# B&R Automation Studio project HealthCareDemo (part 3)

#### SemMan.cpp - SemMan Implementation
```cpp
#include "SemMan.hpp"

RouterSem::RouterSem(UDINT semaphore){
    this->_sem = semaphore;
}

//destructor
RouterSem::~RouterSem(){
    this->_type_id = rl6dNO_TYPE_ID;
}

UDINT RouterSem::get_type_id(void){
    return this->_type_id;
}
UDINT RouterSem::get_semaphore_ident(void){
    return this->_sem;
}
void RouterSem::set_delete(void){
    this->_delete = 1;
}
bool RouterSem::get_delete(void){
    return this->_delete;
}
bool RouterSem::sem_acquire(void){
    return SemAcquire(this->_sem) == ERR_OK;
}
void RouterSem::sem_release(void){
    SemRelease(this->_sem);
}
std::shared_ptr<RouterSem> RouterSem::get_shared_ptr(){
    return shared_from_this();
}

RouterSemBase::RouterSemBase(std::shared_ptr<RouterSem> router_sem){
    this->_router_semaphore = router_sem;
}

//destructor
RouterSemBase::~RouterSemBase(){
    this->_router_semaphore->set_delete();
}

bool RouterSemBase::sem_acquire(void){
    return this->_router_semaphore->sem_acquire();
}
void RouterSemBase::sem_release(void){
    this->_router_semaphore->sem_release();
}

SemMan::SemMan(){
    std::memset(&this->_create_semaphore, 0, sizeof(this->_create_semaphore));
    std::memset(&this->_delete_semaphore, 0, sizeof(this->_delete_semaphore));
}

//destructor
SemMan::~SemMan(){
    this->_type_id = rl6dNO_TYPE_ID;
}

// methods
UDINT SemMan::get_type_id(){
    return this->_type_id;
}
void SemMan::set_create_sem(){
    this->_cmd.create_sem = 1;
}
void SemMan::reset_create_sem(){
    this->_cmd.create_sem = 0;
}
std::shared_ptr<RouterSem> SemMan::get_created_sem(){
    return this->_created_semaphore;
}
bool SemMan::get_cmd_ready(){
    return this->_status.cmd_ready;
}
bool SemMan::get_done(){
    return this->_status.done;
}
bool SemMan::sem_acquire(){
    return SemAcquire(this->_sem) == ERR_OK;
}
void SemMan::sem_release(){
    SemRelease(this->_sem);
}
bool SemMan::get_initialized(){
    return this->_init_done;
}
void SemMan::cyclic(){

    switch(this->_state){

        case STATE_START:

            this->_create_semaphore.enable = 0;
            if(this->_create_semaphore.status == ERR_FUB_ENABLE_FALSE){
                this->_state = STATE_INIT;
            }

            break;

        case STATE_INIT:

            this->_create_semaphore.maxCount = 1;
            this->_create_semaphore.initCount = 1;
            this->_create_semaphore.enable = 1;
            if(this->_create_semaphore.status == ERR_OK){
                this->_sem = this->_create_semaphore.ident;
                this->_create_semaphore.enable = 0;
                this->_status.cmd_ready = 1;
                this->_init_done = 1;
                this->_state = STATE_IDLE;
            }
            else if(!((this->_create_semaphore.status == ERR_FUB_ENABLE_FALSE)||(this->_create_semaphore.status == ERR_FUB_BUSY))){
                this->_create_semaphore.enable = 0;
            }

            break;

        case STATE_IDLE:

            if(this->_cmd.delete_all){
                this->_status.cmd_ready = 0;
                // start deleting all semaphores to prepare for destruction of object
                this->_sem_iterator = this->_semaphores.begin();
                this->_state = STATE_DELETE_ALL_SEM_NEXT;
            }
            else if(this->_cmd.create_sem){
                this->_status.cmd_ready = 0;
                this->_state = STATE_CREATE_SEM;
            }
            else{
                auto it = std::find_if(this->_semaphores.begin(), this->_semaphores.end(), [](std::shared_ptr<RouterSem> i){return i->get_delete();});
                if(it != this->_semaphores.end()){
                    this->_status.cmd_ready = 0;
                    this->_sem_iterator = it;
                    std::shared_ptr<RouterSem> sem = *it;
                    this->_delete_semaphore.ident = sem->get_semaphore_ident();
                    this->_delete_semaphore.enable = 1;
                    this->_state = STATE_DELETE_SEM;
                }
            }

            break;

        case STATE_CREATE_SEM:

            this->_create_semaphore.enable = 1;

            if(this->_create_semaphore.status == ERR_OK){
                std::shared_ptr<RouterSem> new_sem (new RouterSem(this->_create_semaphore.ident));
                this->_created_semaphore = new_sem;
                this->_semaphores.push_back(new_sem);
                this->_create_semaphore.enable = 0;
                this->_status.done = 1;
                this->_state = STATE_CREATE_SEM_DONE;
            }
            else if(!((this->_create_semaphore.status == ERR_FUB_ENABLE_FALSE)||(this->_create_semaphore.status == ERR_FUB_BUSY))){
                this->_create_semaphore.enable = 0;
            }

            break;

        case STATE_CREATE_SEM_DONE:

            if(!this->_cmd.create_sem){
                this->_status.done = 0;
                this->_created_semaphore.reset();
                this->_status.cmd_ready = 1;
                this->_state = STATE_IDLE;
            }

            break;

        case STATE_DELETE_SEM:

            if(!((this->_delete_semaphore.status == ERR_FUB_ENABLE_FALSE)||(this->_delete_semaphore.status == ERR_FUB_BUSY))){
                this->_delete_semaphore.enable = 0;
                this->_semaphores.erase(this->_sem_iterator);
                this->_status.cmd_ready = 1;
                this->_state = STATE_IDLE;
            }

            break;

        case STATE_DELETE_ALL_SEM:

            if(!((this->_delete_semaphore.status == ERR_FUB_ENABLE_FALSE)||(this->_delete_semaphore.status == ERR_FUB_BUSY))){
                this->_delete_semaphore.enable = 0;
                this->_sem_iterator++;
                this->_state = STATE_DELETE_ALL_SEM_NEXT;
            }

            break;

        case STATE_DELETE_ALL_SEM_NEXT:

            if(this->_sem_iterator < this->_semaphores.end()){
                std::shared_ptr<RouterSem> sem = *this->_sem_iterator;
                this->_delete_semaphore.ident = sem->get_semaphore_ident();
                this->_delete_semaphore.enable = 1;
                this->_state = STATE_DELETE_ALL_SEM;
            }
            else{
                this->_delete_semaphore.ident = this->_sem;
                this->_delete_semaphore.enable = 1;
                this->_state = STATE_DELETE_ALL_SEM_LAST;
            }

            break;

        case STATE_DELETE_ALL_SEM_LAST:
            if(!((this->_delete_semaphore.status == ERR_FUB_ENABLE_FALSE)||(this->_delete_semaphore.status == ERR_FUB_BUSY))){
                this->_delete_semaphore.enable = 0;
                this->_semaphores.clear();
                this->_status.done = 1;
                this->_state = STATE_DELETE_ALL_SEM_DONE;
            }
            break;

        case STATE_DELETE_ALL_SEM_DONE:
            //At this point, the object must be destroyed
            break;

    }

    SemCreate(&this->_create_semaphore);
    SemDelete(&this->_delete_semaphore);

}

SemManBase::SemManBase() = default;

//destructor
SemManBase::~SemManBase() = default;

// methods
void SemManBase::set_create_sem(){
    this->_semaphore_manager.set_create_sem();
}
void SemManBase::reset_create_sem(){
    this->_semaphore_manager.reset_create_sem();
}
std::shared_ptr<RouterSem> SemManBase::get_created_sem(){
    return this->_semaphore_manager.get_created_sem();
}
bool SemManBase::get_sem_cmd_ready(){
    return this->_semaphore_manager.get_cmd_ready();
}
bool SemManBase::get_sem_done(){
    return this->_semaphore_manager.get_done();
}
bool SemManBase::sem_acquire(){
    return this->_semaphore_manager.sem_acquire();
}
void SemManBase::sem_release(){
    this->_semaphore_manager.sem_release();
}
```

#### Destination.cpp - Destination Implementation
```cpp
#include "Destination.hpp"

Destination::Destination(std::string name, std::shared_ptr<RouterSem> router_sem): RouterSemBase{router_sem}{
    this->_name = name;
}
Destination::Destination(std::string name, std::shared_ptr<RouterSem> router_sem, rl6dPositionType position): RouterSemBase{router_sem}{
    this->_name = name;
    this->_position = position;
}
Destination::Destination(std::string name, std::shared_ptr<RouterSem> router_sem, rl6dPositionType position, std::shared_ptr<Path> path_in, std::shared_ptr<Path> path_out): RouterSemBase{router_sem}{
    this->_name = name;
    this->_position = position;
    this->_path_in = path_in;
    this->_path_out = path_out;
}

//destructor
Destination::~Destination(){
    this->_type_id = rl6dNO_TYPE_ID;
}

// methods
UDINT Destination::get_type_id(){
    return this->_type_id;
}
std::string Destination::get_name(){
    return this->_name;
}
rl6dPositionType Destination::get_position(){
    return this->_position;
}
void Destination::set_position(rl6dPositionType position){
    this->_position = position;
}
std::shared_ptr<Path> Destination::get_path_in(){
    return this->_path_in;
}
void Destination::set_path_in(std::shared_ptr<Path> path){
    this->_path_in = path;
}
void Destination::clear_path_in(void){
    this->_path_in.reset();
}
std::shared_ptr<Path> Destination::get_path_out(){
    return this->_path_out;
}
void Destination::set_path_out(std::shared_ptr<Path> path){
    this->_path_out = path;
}
void Destination::clear_path_out(){
    this->_path_out.reset();
}
void Destination::set_waypoint(std::weak_ptr<Waypoint> waypoint){
    this->_waypoint = waypoint;
}
std::weak_ptr<Waypoint> Destination::get_waypoint(){
    return this->_waypoint;
}
void Destination::reset_waypoint(){
    this->_waypoint.reset();
}
std::shared_ptr<Destination> Destination::get_shared_ptr(){
    return shared_from_this();
}
std::shared_ptr<DestinationIf> Destination::create_interface(){
    std::shared_ptr<DestinationIf> destination_if (new DestinationIf);
    this->_interfaces.push_back(destination_if);
    return destination_if;
}
void Destination::add_recovery_position(rl6dPositionType position){
    this->_recovery_positions.push_back(position);
}
std::vector<rl6dPositionType> Destination::get_recovery_positions(){
    return this->_recovery_positions;
}
void Destination::set_shuttle_present(std::weak_ptr<Shuttle> shuttle){
    this->_shuttle = shuttle;
    this->_shuttle_present = 1;
}
void Destination::cyclic(){

    if(this->_shuttle_present){
        if(this->sem_acquire()){
            for(auto & interface : this->_interfaces){
                interface->set_shuttle_present(this->_shuttle);
            }
            this->sem_release();
            this->_shuttle_present = 0;
            this->_shuttle.reset();
        }
    }

    if(this->sem_acquire()){
        auto it = std::find_if(this->_interfaces.begin(), this->_interfaces.end(), [](std::shared_ptr<DestinationIf> i){return i->get_delete();});
            if(it != this->_interfaces.end()){
            this->_interfaces.erase(it);
        }
        this->sem_release();
    }

}
```

#### DestinationIf.cpp - DestinationIf Implementation
```cpp
#include "DestinationIf.hpp"

DestinationIf::DestinationIf() = default;

//destructor
DestinationIf::~DestinationIf(){
    this->_type_id = rl6dNO_TYPE_ID;
}

// methods
UDINT DestinationIf::get_type_id(){
    return this->_type_id;
}
std::shared_ptr<DestinationIf> DestinationIf::get_shared_ptr(){
    return shared_from_this();
}
void DestinationIf::set_shuttle_present(std::weak_ptr<Shuttle> shuttle){
    this->_shuttle = shuttle;
    this->_shuttle_present = 1;
}
bool DestinationIf::shuttle_is_present(void){
    return this->_shuttle_present;
}
void DestinationIf::acknowledge_shuttle(){
    this->_shuttle.reset();
    this->_shuttle_present = 0;
}
std::weak_ptr<Shuttle> DestinationIf::get_shuttle_present(){
    return this->_shuttle;
}
void DestinationIf::set_delete(){
    this->_delete = 1;
}
bool DestinationIf::get_delete(){
    return this->_delete;
}
```

#### Path.cpp - Path Implementation
```cpp
#include "Path.hpp"

Path::Path(std::string name, std::shared_ptr<RouterSem> router_sem) : RouterSemBase{router_sem}{
    this->_name = name;
}

//destructor
Path::~Path(){
    this->_type_id = rl6dNO_TYPE_ID;
}

// methods
UDINT Path::get_type_id(){
    return this->_type_id;
}
void Path::add_position(rl6dPositionType position){
    this->_positions.push_back(position);
}
std::string Path::get_name(){
    return this->_name;
}
std::shared_ptr<Path> Path::get_shared_ptr(){
    return shared_from_this();
}
std::vector<rl6dPositionType> Path::get_positions(){
    return this->_positions;
}
```

#### Waypoint.cpp - Waypoint Implementation
```cpp
#include "Waypoint.hpp"

Waypoint::Waypoint(std::string name, std::shared_ptr<RouterSem> router_sem) : RouterSemBase{router_sem}{
    this->_name = name;
}
Waypoint::Waypoint(std::string name, std::shared_ptr<RouterSem> router_sem, rl6dPositionType position) : RouterSemBase{router_sem}{
    this->_name = name;
    this->_position = position;
}

//destructor
Waypoint::~Waypoint(){
    this->_type_id = rl6dNO_TYPE_ID;
}

// methods
UDINT Waypoint::get_type_id(){
    return this->_type_id;
}
std::string Waypoint::get_name(){
    return this->_name;
}
std::shared_ptr<Waypoint> Waypoint::get_shared_ptr(){
    return shared_from_this();
}
void Waypoint::add_destination(std::shared_ptr<Destination> destination, std::shared_ptr<Path> departure_path){
    WaypointDestination waypoint_destination = {destination, departure_path};
    this->_destinations.push_back(waypoint_destination);
}
std::vector<WaypointDestination> Waypoint::get_destinations(void){
    return this->_destinations;
}
rl6dPositionType Waypoint::get_position(void){
    return this->_position;
}
std::weak_ptr<Waypoint> Waypoint::get_next_waypoint(void){
    return this->_next_waypoint;
}
void Waypoint::set_next_waypoint(std::weak_ptr<Waypoint> waypoint){
    this->_next_waypoint = waypoint;
}
void Waypoint::reset_next_waypoint(void){
    this->_next_waypoint.reset();
}
bool Waypoint::check_destination_accessible(std::shared_ptr<Destination> destination){
    for (auto & accessible_destination : this->_destinations){
        if(accessible_destination.destination == destination){
            return true;
        }
    }
    return false;
}
std::shared_ptr<Path> Waypoint::get_destination_departure_path(std::shared_ptr<Destination> destination){
    std::shared_ptr<Path> path;
    auto it = std::find_if(this->_destinations.begin(), this->_destinations.end(), [destination](WaypointDestination i){return i.destination == destination;});
    if(it != this->_destinations.end()){
        path = it->departure_path;
    }
    return path;
}
```

#### Shuttle.cpp - Shuttle Implementation
```cpp
#include "Shuttle.hpp"
ShuttleRoutePositionGenerator::ShuttleRoutePositionGenerator(){
    std::memset(&this->position, 0, sizeof(this->position));
    this->_previous_destination.reset();
    this->_next_destination.reset();
    this->_route_waypoint.reset();
    this->_current_waypoint.reset();
    this->_departure_path.reset();
}
ShuttleRoutePositionGenerator::ShuttleRoutePositionGenerator(std::shared_ptr<Destination> previous_destination, std::shared_ptr<Destination> next_destination){
    std::memset(&this->position, 0, sizeof(this->position));
    this->_previous_destination = previous_destination;
    this->_next_destination = next_destination;
    this->_route_waypoint.reset();
    this->_current_waypoint.reset();
    this->_departure_path.reset();
}
ShuttleRoutePositionGenerator::ShuttleRoutePositionGenerator(std::shared_ptr<Destination> previous_destination, std::shared_ptr<Destination> next_destination, std::weak_ptr<Waypoint> route_waypoint){
    std::memset(&this->position, 0, sizeof(this->position));
    this->_previous_destination = previous_destination;
    this->_next_destination = next_destination;
    this->_route_waypoint = route_waypoint;
    this->_current_waypoint.reset();
    this->_departure_path.reset();
}

ShuttleRoutePositionGenerator::~ShuttleRoutePositionGenerator() = default;

set_path_status_enum ShuttleRoutePositionGenerator::_set_path(std::shared_ptr<Path> path){
    this->_path = path;
    if(this->_path){
        if(this->_path->sem_acquire()){
            this->_path_positions = this->_path->get_positions();
            this->_path->sem_release();
            this->_path_iterator = this->_path_positions.begin();
            if(this->_path_iterator == this->_path_positions.end()){
                return set_path_status_invalid;
            }
            else{
                return set_path_status_valid;
            }
        }
        else{
            return set_path_status_wait_sem;
        }
    }
    else{
        return set_path_status_invalid;
    }
}

bool ShuttleRoutePositionGenerator::operator++(int){

    std::shared_ptr<Waypoint> waypoint;
    rl6dPositionType position;

    if(this->_phase == ROUTED_MOVE_PHASE_EXIT_DEST_START){
        //PHASE_EXIT_DEST_START: Attempt to get the exit path

        if(this->_previous_destination){
            this->_exit_path_status = this->_set_path(this->_previous_destination->get_path_out());
            if(this->_exit_path_status == set_path_status_valid){
                this->position.X = this->_path_iterator->X;
                this->position.Y = this->_path_iterator->Y;
                this->_path_iterator++;
                this->_phase = ROUTED_MOVE_PHASE_EXIT_DEST;
                this->event.path = this->_path;
                this->event.waypoint.reset();
                this->event.event = ROUTED_MOVE_EVENT_PATH_START;
                return true;
            }
            else if(this->_exit_path_status == set_path_status_wait_sem){
                this->event.path.reset();
                this->event.waypoint.reset();
                this->event.event = ROUTED_MOVE_EVENT_NONE;
                return false;
            }
        }
        this->_phase = ROUTED_MOVE_PHASE_WAYPOINT_START; //There is no exit path

    }
    if(this->_phase == ROUTED_MOVE_PHASE_EXIT_DEST){
        //PHASE_EXIT_DEST: Follow the exit path

        if(this->_path_iterator < this->_path_positions.end()){
            this->position.X = this->_path_iterator->X;
            this->position.Y = this->_path_iterator->Y;
            this->_path_iterator++;
            this->event.path.reset();
            this->event.waypoint.reset();
            this->event.event = ROUTED_MOVE_EVENT_NONE;
            return true;
        }
        this->_phase = ROUTED_MOVE_PHASE_WAYPOINT_START; //There are no points left on the exit path

    }
    if(this->_phase == ROUTED_MOVE_PHASE_WAYPOINT_START){
        //PHASE_WAYPOINT_START: Attempt to get the waypoint

        if(!this->_route_waypoint.expired()){
            this->_current_waypoint = this->_route_waypoint;
        }
        else if(this->_previous_destination){
            this->_current_waypoint = this->_previous_destination->get_waypoint();
        }
        if(!this->_current_waypoint.expired()){
            waypoint = this->_current_waypoint.lock();
            position = waypoint->get_position();
            this->position.X = position.X;
            this->position.Y = position.Y;
            this->_phase = ROUTED_MOVE_PHASE_WAYPOINT;
            this->event.path.reset();
            this->event.waypoint = this->_current_waypoint;
            this->event.event = ROUTED_MOVE_EVENT_WAYPOINT;
            return true;
        }
        this->_phase = ROUTED_MOVE_PHASE_ENTER_DEST_START; //There is no waypoint

    }
    if(this->_phase == ROUTED_MOVE_PHASE_WAYPOINT){
        //PHASE_WAYPOINT: Follow waypoints

        if(!this->_current_waypoint.expired()){
            waypoint = this->_current_waypoint.lock();
            if(waypoint->sem_acquire()){
                bool destination_accessible = waypoint->check_destination_accessible(this->_next_destination);
                if(destination_accessible){
                    this->_departure_path = waypoint->get_destination_departure_path(this->_next_destination);
                    waypoint->sem_release();
                    this->_phase = ROUTED_MOVE_PHASE_DEPART_WAYPOINT_START;
                }
                else{
                    waypoint->sem_release();
                    this->_current_waypoint = waypoint->get_next_waypoint();
                    if(!this->_current_waypoint.expired()){
                        waypoint = this->_current_waypoint.lock();
                        position = waypoint->get_position();
                        this->position.X = position.X;
                        this->position.Y = position.Y;
                        this->event.path.reset();
                        this->event.waypoint = this->_current_waypoint;
                        this->event.event = ROUTED_MOVE_EVENT_WAYPOINT;
                        return true;
                    }
                }
            }
            else{
                this->event.path.reset();
                this->event.waypoint.reset();
                this->event.event = ROUTED_MOVE_EVENT_NONE;
                return false;
            }
        }
        else{
            //Something went wrong here - the waypoint should not be expired
            this->_phase = ROUTED_MOVE_PHASE_ENTER_DEST_START;
        }

    }
    if(this->_phase == ROUTED_MOVE_PHASE_DEPART_WAYPOINT_START){
        //PHASE_DEPART_WAYPOINT_START: Attempt to get the departure path

        this->_departure_path_status = this->_set_path(this->_departure_path);
        if(this->_departure_path_status == set_path_status_valid){
            this->position.X = this->_path_iterator->X;
            this->position.Y = this->_path_iterator->Y;
            this->_path_iterator++;
            this->_phase = ROUTED_MOVE_PHASE_DEPART_WAYPOINT;
            this->event.path = this->_path;
            this->event.waypoint.reset();
            this->event.event = ROUTED_MOVE_EVENT_PATH_START;
            return true;
        }
        else if(this->_departure_path_status == set_path_status_wait_sem){
            this->event.path.reset();
            this->event.waypoint.reset();
            this->event.event = ROUTED_MOVE_EVENT_NONE;
            return false;
        }
        this->_phase = ROUTED_MOVE_PHASE_ENTER_DEST_START; //There is no departure path

    }
    if(this->_phase == ROUTED_MOVE_PHASE_DEPART_WAYPOINT){
        //PHASE_DEPART_WAYPOINT_START: Follow the departure path

        if(this->_departure_path_status == set_path_status_valid){
            if(this->_path_iterator < this->_path_positions.end()){
                this->position.X = this->_path_iterator->X;
                this->position.Y = this->_path_iterator->Y;
                this->_path_iterator++;
                this->event.path.reset();
                this->event.waypoint.reset();
                this->event.event = ROUTED_MOVE_EVENT_NONE;
                return true;
            }
        }
        this->_phase = ROUTED_MOVE_PHASE_ENTER_DEST_START; //There are no points left on the departure path

    }
    if(this->_phase == ROUTED_MOVE_PHASE_ENTER_DEST_START){
        //ROUTED_MOVE_PHASE_ENTER_DEST_START: Attempt to get the entry path

        this->_entry_path_status = this->_set_path(this->_next_destination->get_path_in());
        if(this->_entry_path_status == set_path_status_valid){
            this->position.X = this->_path_iterator->X;
            this->position.Y = this->_path_iterator->Y;
            this->_path_iterator++;
            this->_phase = ROUTED_MOVE_PHASE_ENTER_DEST;
            this->event.path = this->_path;
            this->event.waypoint.reset();
            this->event.event = ROUTED_MOVE_EVENT_PATH_START;
            return true;
        }
        else if(this->_entry_path_status == set_path_status_wait_sem){
            this->event.path.reset();
            this->event.waypoint.reset();
            this->event.event = ROUTED_MOVE_EVENT_NONE;
            return false;
        }
        this->_phase = ROUTED_MOVE_PHASE_DEST; //There is no entry path

    }
    if(this->_phase == ROUTED_MOVE_PHASE_ENTER_DEST){
        //ROUTED_MOVE_PHASE_ENTER_DEST: Follow the entry path

        if(this->_entry_path_status == set_path_status_valid){
            if(this->_path_iterator < this->_path_positions.end()){
                this->position.X = this->_path_iterator->X;
                this->position.Y = this->_path_iterator->Y;
                this->_path_iterator++;
                this->event.path.reset();
                this->event.waypoint.reset();
                this->event.event = ROUTED_MOVE_EVENT_NONE;
                return true;
            }
        }
        this->_phase = ROUTED_MOVE_PHASE_DEST; //There are no points left on the entry path

    }
    if(this->_phase == ROUTED_MOVE_PHASE_DEST){
        //ROUTED_MOVE_PHASE_DEST: Move to destination

        position = this->_next_destination->get_position();
        this->position.X = position.X;
        this->position.Y = position.Y;
        if(this->_updated_destination){
            this->_previous_destination = this->_next_destination;
            this->_next_destination = this->_updated_destination;
            this->_updated_destination.reset();
            this->_phase = ROUTED_MOVE_PHASE_EXIT_DEST_START;
        }
        else{
            this->_done = 1;
            this->_phase = ROUTED_MOVE_PHASE_ARRIVE;
        }
        this->event.path.reset();
        this->event.waypoint.reset();
        this->event.event = ROUTED_MOVE_EVENT_NONE;
        return true;

    }

    return false;

}

void ShuttleRoutePositionGenerator::update_destination(std::shared_ptr<Destination> destination){
    if(this->_phase < ROUTED_MOVE_PHASE_DEPART_WAYPOINT_START){ //We have not yet left for the current destination
        this->_next_destination = destination;
    }
    else{
        this->_updated_destination = destination;
    }
}

void ShuttleRoutePositionGenerator::update_destination(std::shared_ptr<Destination> destination, std::weak_ptr<Waypoint> waypoint){
    if(!waypoint.expired()){
        this->_route_waypoint = waypoint;
    }
    if(this->_phase < ROUTED_MOVE_PHASE_DEPART_WAYPOINT_START){ //We have not yet left for the current destination
        this->_next_destination = destination;
    }
    else{
        this->_updated_destination = destination;
    }
}

routed_move_phase_enum ShuttleRoutePositionGenerator::get_phase(){
    return this->_phase;
}
bool ShuttleRoutePositionGenerator::get_done(){
    return this->_done;
}

Shuttle::Shuttle(Mc6DShuttleType shuttle, std::shared_ptr<RouterSem> router_sem, UDINT user_data_size, UINT shuttle_id) : RouterSemBase{router_sem}{
    std::memset(&this->_move_in_plane, 0, sizeof(this->_move_in_plane));
    this->_shuttle = shuttle;
    this->_move_in_plane.Shuttle = &this->_shuttle;
    this->_move_in_plane.Parameters.Mode = mcACP6D_MOVE_ABSOLUTE;
    this->_user_data = std::unique_ptr<char[]>(new char[user_data_size]);
    std::memset(this->_user_data.get(), 0, user_data_size);
    this->_user_data_size = user_data_size;
    this->_shuttle_id = shuttle_id;
}

//destructor
Shuttle::~Shuttle(){
    this->_type_id = rl6dNO_TYPE_ID;
}

// methods
UDINT Shuttle::get_type_id(){
    return this->_type_id;
}
UINT Shuttle::get_shuttle_id(){
    return this->_shuttle_id;
}
Mc6DShuttleType* Shuttle::get_shuttle_reference(){
    return &this->_shuttle;
}
std::shared_ptr<Destination> Shuttle::get_current_destination(){
    return this->_next_destination;
}
std::shared_ptr<Destination> Shuttle::get_previous_destination(){
    return this->_previous_destination;
}
void Shuttle::clear_previous_destination(){
    this->_previous_destination.reset();
}
std::shared_ptr<ShuttleIf> Shuttle::create_interface(){
    std::shared_ptr<ShuttleIf> shuttle_if (new ShuttleIf);
    this->_interfaces.push_back(shuttle_if);
    return shuttle_if;
}
std::shared_ptr<Shuttle> Shuttle::get_shared_ptr(){
    return shared_from_this();
}
ReadUserDataResult Shuttle::read_user_data(){
    ReadUserDataResult result = {this->_user_data.get(), this->_user_data_size};
    return result;
}
UDINT Shuttle::write_user_data(char* value, UDINT size){
    if(size < this->_user_data_size){
        std::memcpy(this->_user_data.get(), value, size);
        return size;
    }
    else{
        std::memcpy(this->_user_data.get(), value, this->_user_data_size);
        return this->_user_data_size;
    }
}
bool Shuttle::_update_interfaces(){
    if(this->_current_interface){
        if(this->_interfaces.empty()){ //The current interface is defined, but no interfaces are being used
            this->_current_interface.reset();
            return 1; //Indicate that the interface has changed
        }
        else if(this->_current_interface != this->_interfaces.back()){ //A newer interface is available
            std::shared_ptr<ShuttleIf> interface = this->_current_interface;
            interface->reset_move_active();
            interface->set_aborted();
            this->_current_interface = this->_interfaces.back();
            return 1; //Indicate that the interface has changed
        }
    }
    else if(!this->_interfaces.empty()){ //No interface is defined, but an interface is available
        this->_current_interface = this->_interfaces.back();
        return 1; //Indicate that the interface has changed
    }
    return 0; //Indicate that the interface has not changed
}

void Shuttle::_log_event(RoutedMoveEvent event){

    switch(event.event){

        case ROUTED_MOVE_EVENT_NONE:

            break;

        case ROUTED_MOVE_EVENT_PATH_START:
            log_path_start(this->get_shuttle_id(), this->_route_position_generator.event.path->get_name());
            break;

        case ROUTED_MOVE_EVENT_WAYPOINT:
            log_waypoint_move(this->get_shuttle_id(), this->_route_position_generator.event.waypoint.lock()->get_name());
            break;

    }

    return;

}

void Shuttle::cyclic(){

    rl6dPositionType position;

    switch(this->_state){

        case STATE_IDLE:

            if(this->_update_interfaces()){
                if(this->_current_interface){
                    this->_move_in_plane.Parameters.Velocity = this->_current_interface->get_velocity();
                    this->_move_in_plane.Parameters.Acceleration = this->_current_interface->get_acceleration();
                    this->_current_interface->set_move_active();
                    this->_next_destination = this->_current_interface->get_destination();
                    if(this->_current_interface->get_destination_direct_command()){
                        position = this->_next_destination->get_position();
                        this->_move_in_plane.Parameters.Position.X = position.X;
                        this->_move_in_plane.Parameters.Position.Y = position.Y;
                        this->_move_in_plane.Execute = 1;
                        log_direct_move_start(this->get_shuttle_id(), this->_next_destination->get_name());
                        this->_state = STATE_DIRECT_MOVE;
                    }
                    else if(this->_current_interface->get_destination_command()){
                        this->_optional_waypoint = this->_current_interface->get_waypoint();
                        this->_route_position_generator = ShuttleRoutePositionGenerator(this->_previous_destination, this->_next_destination, this->_optional_waypoint);
                        if(this->_route_position_generator++){
                            this->_move_in_plane.Parameters.Position.X = _route_position_generator.position.X;
                            this->_move_in_plane.Parameters.Position.Y = _route_position_generator.position.Y;
                            this->_move_in_plane.Execute = 1;
                            if(this->_optional_waypoint.expired()){
                                log_routed_move_start(this->get_shuttle_id(), this->_next_destination->get_name());
                            }
                            else{
                                log_routed_move_waypoint(this->get_shuttle_id(), this->_next_destination->get_name(), this->_optional_waypoint.lock()->get_name());
                            }
                            this->_log_event(this->_route_position_generator.event);
                            this->_state = STATE_ROUTED_MOVE;
                        }
                        else{
                            this->_state = STATE_ROUTED_MOVE_START;
                        }
                    }
                }
            }

            break;

        case STATE_ROUTED_MOVE_START:

            if(this->_route_position_generator++){
                this->_move_in_plane.Parameters.Position.X = _route_position_generator.position.X;
                this->_move_in_plane.Parameters.Position.Y = _route_position_generator.position.Y;
                this->_move_in_plane.Execute = 1;
                if(this->_optional_waypoint.expired()){
                    log_routed_move_start(this->get_shuttle_id(), this->_next_destination->get_name());
                }
                else{
                    log_routed_move_waypoint(this->get_shuttle_id(), this->_next_destination->get_name(), this->_optional_waypoint.lock()->get_name());
                }
                this->_log_event(this->_route_position_generator.event);
                this->_state = STATE_ROUTED_MOVE;
            }

            break;

        case STATE_ROUTED_MOVE:

            if(this->_move_in_plane.Done){
                this->_move_in_plane.Execute = 0;
                if(this->_route_position_generator.get_done()){
                    log_destination_arrival(this->get_shuttle_id(), this->_next_destination->get_name());
                    if(this->_current_interface){
                        this->_current_interface->set_move_done();
                    }
                    std::weak_ptr<Shuttle> reference = shared_from_this();
                    this->_next_destination->set_shuttle_present(reference);
                    this->_previous_destination = this->_next_destination;
                    this->_next_destination.reset();
                    this->_state = STATE_IDLE;
                }
                else{
                    this->_state = STATE_ROUTED_MOVE_NEXT;
                }
            }
            else if(this->_move_in_plane.Error){
                log_sh_error(this->get_shuttle_id(), this->_move_in_plane.ErrorID);
                this->_move_in_plane.Execute = 0;
                this->_current_interface->set_error(this->_move_in_plane.ErrorID);
                this->_state = STATE_IDLE;
            }

            break;

        case STATE_ROUTED_MOVE_NEXT:

            if(this->_update_interfaces()){
                if(this->_current_interface){
                    this->_move_in_plane.Parameters.Velocity = this->_current_interface->get_velocity();
                    this->_move_in_plane.Parameters.Acceleration = this->_current_interface->get_acceleration();
                    this->_current_interface->set_move_active();
                    this->_next_destination = this->_current_interface->get_destination();
                    this->_route_position_generator.update_destination(this->_next_destination);
                    log_destination_update(this->get_shuttle_id(), this->_next_destination->get_name());
                }
            }
            if(this->_route_position_generator++){
                this->_move_in_plane.Parameters.Position.X = _route_position_generator.position.X;
                this->_move_in_plane.Parameters.Position.Y = _route_position_generator.position.Y;
                this->_move_in_plane.Execute = 1;
                this->_log_event(this->_route_position_generator.event);
                this->_state = STATE_ROUTED_MOVE;
            }

            break;

        case STATE_DIRECT_MOVE:

            if(this->_move_in_plane.Done){
                this->_move_in_plane.Execute = 0;
                log_destination_arrival(this->get_shuttle_id(), this->_next_destination->get_name());
                if(this->_current_interface){
                    this->_current_interface->set_move_done();
                }
                std::weak_ptr<Shuttle> reference = shared_from_this();
                this->_next_destination->set_shuttle_present(reference);
                this->_previous_destination = this->_next_destination;
                this->_next_destination.reset();
                this->_state = STATE_IDLE;
            }
            else if(this->_move_in_plane.Error){
                log_sh_error(this->get_shuttle_id(), this->_move_in_plane.ErrorID);
                this->_move_in_plane.Execute = 0;
                if(this->_current_interface){
                    this->_current_interface->set_error(this->_move_in_plane.ErrorID);
                }
                this->_state = STATE_IDLE;
            }

            break;

    }

    if(this->sem_acquire()){
        auto it_delete = std::find_if(this->_interfaces.begin(), this->_interfaces.end(), [](std::shared_ptr<ShuttleIf> i){return i->get_delete();});
        if(it_delete != this->_interfaces.end()){
            this->_interfaces.erase(it_delete);
        }
        //Delete any invalid interfaces
        auto it_invalid = std::find_if(this->_interfaces.begin(), this->_interfaces.end(), [](std::shared_ptr<ShuttleIf> i){return (i->get_type_id() != rl6dSHUTTLE_IF_TYPE_ID);});
        if(it_invalid != this->_interfaces.end()){
            this->_interfaces.erase(it_invalid);
        }
        this->sem_release();
    }

    MC_BR_MoveInPlane_Acp6D(&this->_move_in_plane);

}
```

#### ShuttleIf.cpp - DestinationIf Implementation
```cpp
#include "ShuttleIf.hpp"

ShuttleIf::ShuttleIf() = default;

//destructor
ShuttleIf::~ShuttleIf(){
    this->_type_id = rl6dNO_TYPE_ID;
}

// methods
UDINT ShuttleIf::get_type_id(){
    return this->_type_id;
}
void ShuttleIf::set_destination(std::shared_ptr<Destination> destination, REAL velocity, REAL acceleration){
    this->_destination = destination;
    this->_velocity = velocity;
    this->_acceleration = acceleration;
    this->_move_destination = 1;
}
bool ShuttleIf::get_destination_command(){
    return this->_move_destination;
}
void ShuttleIf::set_destination_direct(std::shared_ptr<Destination> destination, REAL velocity, REAL acceleration){
    this->_destination = destination;
    this->_velocity = velocity;
    this->_acceleration = acceleration;
    this->_move_destination_direct = 1;
}
bool ShuttleIf::get_destination_direct_command(){
    return this->_move_destination_direct;
}
std::shared_ptr<Destination> ShuttleIf::get_destination(){
    return this->_destination;
}
void ShuttleIf::set_aborted(){
    this->_aborted = 1;
}
bool ShuttleIf::get_aborted(){
    return this->_aborted;
}
void ShuttleIf::set_error(DINT error){
    this->_error = 1;
    this->_error_id = error;
}
bool ShuttleIf::get_error(){
    return this->_error;
}
DINT ShuttleIf::get_error_id(){
    return this->_error_id;
}
void ShuttleIf::set_move_done(){
    this->_move_done = 1;
}
bool ShuttleIf::get_move_done(){
    return this->_move_done;
}
void ShuttleIf::set_move_active(){
    this->_move_active = 1;
}
void ShuttleIf::reset_move_active(){
    this->_move_active = 0;
}
bool ShuttleIf::get_move_active(){
    return this->_move_active;
}
void ShuttleIf::set_delete(){
    this->_delete = 1;
}
bool ShuttleIf::get_delete(){
    return this->_delete;
}
REAL ShuttleIf::get_velocity(){
    return this->_velocity;
}
REAL ShuttleIf::get_acceleration(){
    return this->_acceleration;
}
std::shared_ptr<ShuttleIf> ShuttleIf::get_shared_ptr(){
    return shared_from_this();
}
```

#### rl6dRouterMan.cpp - rl6dRouter Implementation
```cpp
#include "Router.hpp"

uint32_t bur_heap_size = rl6dHEAP_SIZE;

extern "C" _BUR_PUBLIC void rl6dRouterMan(struct rl6dRouterMan* inst){

    if(inst == nullptr){
        return;
    }

    Router* r;
    DINT error;

    enum state{
        state_idle,
        state_active,
        state_error
    };

    switch(inst->Internal.State){

        case state_idle:

            if(inst->Enable){
                inst->Busy = 1;
                if(inst->UserDataSize > 0){
                    inst->Router.Ident = reinterpret_cast<std::uintptr_t>(new Router(inst->Assembly, inst->UserDataSize));
                    inst->Active = 1;
                    inst->Internal.State = state_active;
                }
                else{
                    inst->ErrorID = rl6dERR_USER_DATA_SIZE_ZERO;
                    inst->Error = 1;
                    inst->Internal.State = state_error;
                }
            }

            break;

        case state_active:

            error = check_router_reference(&inst->Router);
            if(error == ERR_OK){
                r = reinterpret_cast<Router*>(inst->Router.Ident);
                r->cyclic();
                if(!inst->Enable){
                    inst->Active = 0;
                    inst->Router.Ident = 0;
                    delete r;
                    inst->Busy = 0;
                    inst->Internal.State = state_idle;
                    }
            }
            else{
                inst->Active = 0;
                inst->ErrorID = error;
                inst->Error = 1;
                inst->Internal.State = state_error;
            }

            break;

        case state_error:

            if(!inst->Enable){
                error = check_router_reference(&inst->Router);
                if(error == ERR_OK){
                    r = reinterpret_cast<Router*>(inst->Router.Ident);
                    delete r;
                }
                inst->Router.Ident = 0;
                inst->ErrorID = ERR_OK;
                inst->Error = 0;
                inst->Busy = 0;
                inst->Internal.State = state_idle;
            }

            break;

    }

    //TODO: Allow for cleanup of semaphores before router deletion

}
```

#### rl6dRouterAddPathFromData.cpp - rl6dRouterAddPathFromData Implementation
```cpp
#include "Router.hpp"

extern "C" _BUR_PUBLIC void rl6dRouterAddPathFromData(struct rl6dRouterAddPathFromData* inst){

    if(inst == nullptr){
        return;
    }

    Router* r;
    RouterSem* router_sem;
    std::shared_ptr<Path> p;
    rl6dPositionType* position;
    DINT error;

    enum state{
        state_idle,
        state_create_sem_start,
        state_create_sem_end,
        state_add_positions,
        state_done,
        state_error
    };

    switch(inst->Internal.State){

        case state_idle:

            if(inst->Execute){
                inst->Busy = 1;
                inst->Internal.State = state_create_sem_start;
            }

            break;

        case state_create_sem_start:

            error = check_router_reference(inst->Router);
            if(error == ERR_OK){
                if(inst->DataSize % sizeof(rl6dPositionType) != 0){
                    error = rl6dERR_DATA_ALIGNMENT;
                }
            }
            if(error == ERR_OK){
                if(inst->Name[0] == 0){
                    error = rl6dERR_NO_OBJ_NAME;
                }
            }
            if(error == ERR_OK){
                r = reinterpret_cast<Router*>(inst->Router->Ident);
                if(r->get_initialized()){
                    if(r->sem_acquire()){
                        if(r->get_sem_cmd_ready()){
                            r->set_create_sem();
                            inst->Internal.State = state_create_sem_end;
                        }
                        else{
                            r->sem_release();
                        }
                    }
                }
            }
            else{
                inst->ErrorID = error;
                inst->Error = 1;
                inst->Internal.State = state_error;
            }
            break;

        case state_create_sem_end:

            error = check_router_reference(inst->Router);
            if(error == ERR_OK){
                r = reinterpret_cast<Router*>(inst->Router->Ident);
                if(r->get_sem_done()){
                    inst->Internal.Reference = reinterpret_cast<std::uintptr_t>(r->get_created_sem().get());
                    r->reset_create_sem();
                    r->sem_release();
                    inst->Internal.State = state_add_positions;
                }
            }
            else{
                inst->ErrorID = error;
                inst->Error = 1;
                inst->Internal.State = state_error;
            }

            break;

        case state_add_positions:

            error = check_router_reference(inst->Router);
            if(error == ERR_OK){
                error = check_router_sem_reference(inst->Internal.Reference);
            }
            if(error == ERR_OK){
                if(inst->DataSize % sizeof(rl6dPositionType) != 0){
                    error = rl6dERR_DATA_ALIGNMENT;
                }
            }
            if(error == ERR_OK){
                if(inst->Name[0] == 0){
                    error = rl6dERR_NO_OBJ_NAME;
                }
            }
            if(error == ERR_OK){
                r = reinterpret_cast<Router*>(inst->Router->Ident);
                if(r->acquire_path_semaphore()){
                    router_sem = reinterpret_cast<RouterSem*>(inst->Internal.Reference);
                    try{
                        p = r->create_path(inst->Name, router_sem->get_shared_ptr());
                    }
                    catch (const std::invalid_argument& ia) {
                        inst->ErrorID = rl6dERR_OBJ_NAME_EXISTS;
                        inst->Error = 1;
                        inst->Internal.State = state_error;
                        r->release_path_semaphore();
                        router_sem->set_delete();
                        return;
                    }
                    for(UDINT offset = 0; offset < inst->DataSize; offset += sizeof(rl6dPositionType)){
                        position = reinterpret_cast<rl6dPositionType*>(inst->DataAddress + offset);
                        p->add_position(*position);
                    }
                    inst->Path.Ident = reinterpret_cast<std::uintptr_t>(p.get());
                    r->release_path_semaphore();
                    inst->Done = 1;
                    inst->Internal.State = state_done;
                }
            }
            else{
                inst->ErrorID = error;
                inst->Error = 1;
                if(check_router_sem_reference(inst->Internal.Reference) == ERR_OK){
                    router_sem = reinterpret_cast<RouterSem*>(inst->Internal.Reference);
                    router_sem->set_delete();
                }
                inst->Internal.State = state_error;
            }

            break;

        case state_done:

            if(!inst->Execute){
                inst->Done = 0;
                inst->Path.Ident = 0;
                inst->Busy = 0;
                inst->Internal.State = state_idle;
            }

            break;

        case state_error:

            if(!inst->Execute){
                inst->ErrorID = ERR_OK;
                inst->Error = 0;
                inst->Busy = 0;
                inst->Internal.State = state_idle;
            }

            break;

    }

}
```

#### rl6dRouterAddDestination.cpp - rl6dRouterAddDestination Implementation
```cpp
#include "Router.hpp"

extern "C" _BUR_PUBLIC void rl6dRouterAddDestination(struct rl6dRouterAddDestination* inst){

    if(inst == nullptr){
        return;
    }

    Router* r;
    RouterSem* router_sem;
    std::shared_ptr<Destination> destination;
    Path* p;
    std::shared_ptr<Path> entry_path;
    std::shared_ptr<Path> exit_path;
    DINT error;

    enum state{
        state_idle,
        state_create_sem_start,
        state_create_sem_end,
        state_create_destination,
        state_done,
        state_error
    };

    switch(inst->Internal.State){

        case state_idle:

            if(inst->Execute){
                inst->Busy = 1;
                inst->Internal.State = state_create_sem_start;
            }

            break;

        case state_create_sem_start:

            error = check_router_reference(inst->Router);
            if(error == ERR_OK){
                if(inst->Name[0] == 0){
                    error = rl6dERR_NO_OBJ_NAME;
                }
            }
            if((error == ERR_OK) && (inst->EntryPath != nullptr)){
                error = check_path_reference(inst->EntryPath);
            }
            if((error == ERR_OK) && (inst->ExitPath != nullptr)){
                error = check_path_reference(inst->ExitPath);
            }
            if(error == ERR_OK){
                r = reinterpret_cast<Router*>(inst->Router->Ident);
                if(r->get_initialized()){
                    if(r->sem_acquire()){
                        if(r->get_sem_cmd_ready()){
                            r->set_create_sem();
                            inst->Internal.State = state_create_sem_end;
                        }
                        else{
                            r->sem_release();
                        }
                    }
                }
            }
            else{
                inst->ErrorID = error;
                inst->Error = 1;
                inst->Internal.State = state_error;
            }
            break;

        case state_create_sem_end:

            error = check_router_reference(inst->Router);
            if(error == ERR_OK){
                r = reinterpret_cast<Router*>(inst->Router->Ident);
                if(r->get_sem_done()){
                    inst->Internal.Reference = reinterpret_cast<std::uintptr_t>(r->get_created_sem().get());
                    r->reset_create_sem();
                    r->sem_release();
                    inst->Internal.State = state_create_destination;
                }
            }
            else{
                inst->ErrorID = error;
                inst->Error = 1;
                inst->Internal.State = state_error;
            }

            break;

        case state_create_destination:

            error = check_router_reference(inst->Router);
            if(error == ERR_OK){
            error = check_router_sem_reference(inst->Internal.Reference);
            }
            if(error == ERR_OK){
                if(inst->Name[0] == 0){
                    error = rl6dERR_NO_OBJ_NAME;
                }
            }
            if((error == ERR_OK) && (inst->EntryPath != nullptr)){
                error = check_path_reference(inst->EntryPath);
            }
            if((error == ERR_OK) && (inst->ExitPath != nullptr)){
                error = check_path_reference(inst->ExitPath);
            }
            if(error == ERR_OK){
                r = reinterpret_cast<Router*>(inst->Router->Ident);
                if(r->acquire_destination_semaphore()){
                    router_sem = reinterpret_cast<RouterSem*>(inst->Internal.Reference);
                    if(inst->EntryPath != nullptr){
                        if(inst->EntryPath->Ident){
                            p = reinterpret_cast<Path*>(inst->EntryPath->Ident);
                            if(p->get_type_id() == rl6dPATH_TYPE_ID){
                                entry_path = p->get_shared_ptr();
                            }
                        }
                    }
                    if(inst->ExitPath != nullptr){
                        if(inst->ExitPath->Ident){
                            p = reinterpret_cast<Path*>(inst->ExitPath->Ident);
                            if(p->get_type_id() == rl6dPATH_TYPE_ID){
                                exit_path = p->get_shared_ptr();
                            }
                        }
                    }
                    try{
                        destination = r->create_destination(inst->Name, router_sem->get_shared_ptr(), inst->Position, entry_path, exit_path);
                    }
                    catch (const std::invalid_argument& ia) {
                        inst->ErrorID = rl6dERR_OBJ_NAME_EXISTS;
                        inst->Error = 1;
                        inst->Internal.State = state_error;
                        r->release_destination_semaphore();
                        router_sem->set_delete();
                        return;
                    }
                    inst->Destination.Ident = reinterpret_cast<std::uintptr_t>(destination.get());
                    r->release_destination_semaphore();
                    inst->Done = 1;
                    inst->Internal.State = state_done;
                }
            }
            else{
                inst->ErrorID = error;
                inst->Error = 1;
                if(check_router_sem_reference(inst->Internal.Reference) == ERR_OK){
                    router_sem = reinterpret_cast<RouterSem*>(inst->Internal.Reference);
                    router_sem->set_delete();
                }
                inst->Internal.State = state_error;
            }

            break;

        case state_done:

            if(!inst->Execute){
                inst->Done = 0;
                inst->Destination.Ident = 0;
                inst->Busy = 0;
                inst->Internal.State = 0;
            }

            break;

        case state_error:

            if(!inst->Execute){
                inst->ErrorID = ERR_OK;
                inst->Error = 0;
                inst->Busy = 0;
                inst->Internal.State = state_idle;
            }

            break;

    }

}
```

#### rl6dRouterAddWaypoint.cpp - rl6dRouterAddWaypoint Implementation
```cpp
#include "Router.hpp"

extern "C" _BUR_PUBLIC void rl6dRouterAddWaypoint(struct rl6dRouterAddWaypoint* inst){

    if(inst == nullptr){
        return;
    }

    Router* r;
    RouterSem* router_sem;
    std::shared_ptr<Waypoint> waypoint;
    DINT error;

    enum state{
        state_idle,
        state_create_sem_start,
        state_create_sem_end,
        state_create_waypoint,
        state_done,
        state_error
    };

    switch(inst->Internal.State){

        case state_idle:

            if(inst->Execute){
                inst->Busy = 1;
                inst->Internal.State = state_create_sem_start;
            }

            break;

        case state_create_sem_start:

            error = check_router_reference(inst->Router);
            if(error == ERR_OK){
                if(inst->Name[0] == 0){
                    error = rl6dERR_NO_OBJ_NAME;
                }
            }
            if(error == ERR_OK){
                r = reinterpret_cast<Router*>(inst->Router->Ident);
                if(r->get_initialized()){
                    if(r->sem_acquire()){
                        if(r->get_sem_cmd_ready()){
                            r->set_create_sem();
                            inst->Internal.State = state_create_sem_end;
                        }
                        else{
                            r->sem_release();
                        }
                    }
                }
            }
            else{
                inst->ErrorID = error;
                inst->Error = 1;
                inst->Internal.State = state_error;
            }
            break;

        case state_create_sem_end:

            error = check_router_reference(inst->Router);
            if(error == ERR_OK){
                r = reinterpret_cast<Router*>(inst->Router->Ident);
                if(r->get_sem_done()){
                    inst->Internal.Reference = reinterpret_cast<std::uintptr_t>(r->get_created_sem().get());
                    r->reset_create_sem();
                    r->sem_release();
                    inst->Internal.State = state_create_waypoint;
                }
            }
            else{
                inst->ErrorID = error;
                inst->Error = 1;
                inst->Internal.State = state_error;
            }

            break;

        case state_create_waypoint:

            error = check_router_reference(inst->Router);
            if(error == ERR_OK){
            error = check_router_sem_reference(inst->Internal.Reference);
            }
            if(error == ERR_OK){
                if(inst->Name[0] == 0){
                    error = rl6dERR_NO_OBJ_NAME;
                }
            }
            if(error == ERR_OK){
                r = reinterpret_cast<Router*>(inst->Router->Ident);
                if(r->acquire_waypoint_semaphore()){
                    router_sem = reinterpret_cast<RouterSem*>(inst->Internal.Reference);
                    try{
                        waypoint = r->create_waypoint(inst->Name, router_sem->get_shared_ptr(), inst->Position);
                    }
                    catch (const std::invalid_argument& ia) {
                        inst->ErrorID = rl6dERR_OBJ_NAME_EXISTS;
                        inst->Error = 1;
                        inst->Internal.State = state_error;
                        r->release_waypoint_semaphore();
                        router_sem->set_delete();
                        return;
                    }
                    inst->Waypoint.Ident = reinterpret_cast<std::uintptr_t>(waypoint.get());
                    r->release_waypoint_semaphore();
                    inst->Done = 1;
                    inst->Internal.State = state_done;
                }
            }
            else{
                inst->ErrorID = error;
                inst->Error = 1;
                if(check_router_sem_reference(inst->Internal.Reference) == ERR_OK){
                    router_sem = reinterpret_cast<RouterSem*>(inst->Internal.Reference);
                    router_sem->set_delete();
                }
                inst->Internal.State = state_error;
            }

            break;

        case state_done:

            if(!inst->Execute){
                inst->Done = 0;
                inst->Waypoint.Ident = 0;
                inst->Busy = 0;
                inst->Internal.State = 0;
            }

            break;

        case state_error:

            if(!inst->Execute){
                inst->ErrorID = ERR_OK;
                inst->Error = 0;
                inst->Busy = 0;
                inst->Internal.State = state_idle;
            }

            break;

    }

}
```

#### rl6dPathGetData.cpp - rl6dGetDataFromPath Implementation
```cpp
#include "Router.hpp"

extern "C" _BUR_PUBLIC void rl6dPathGetData(struct rl6dPathGetData* inst){

    if(inst == nullptr){
        return;
    }

    Path* p;
    std::shared_ptr<Path> path;
    DINT error;

    enum state{
        state_idle,
        state_get_data,
        state_done,
        state_error
    };

    switch(inst->Internal.State){

        case state_idle:

            if(inst->Execute){
                inst->Busy = 1;
                inst->Internal.DataAddress = inst->DataAddress;
                inst->Internal.DataSize = inst->DataSize;
                inst->Internal.State = state_get_data;
            }

            break;

        case state_get_data:

            error = check_path_reference(inst->Path);
            if(error == ERR_OK){
                p = reinterpret_cast<Path*>(inst->Path->Ident);
                path = p->get_shared_ptr();
                if(path->sem_acquire()){
                    std::vector<rl6dPositionType> positions = path->get_positions();
                    path->sem_release();
                    UDINT available_size = inst->Internal.DataSize / sizeof(rl6dPositionType);
                    UDINT offset = 0;
                    for(auto & position : positions){
                        if(offset < available_size){
                            rl6dPositionType* array_position = reinterpret_cast<rl6dPositionType*>(inst->Internal.DataAddress + offset*sizeof(rl6dPositionType));
                            *array_position = position;
                            offset++;
                        }
                        else{
                            break;
                        }
                    }
                    inst->PathDataSize = positions.size() * sizeof(rl6dPositionType);
                    inst->Done = 1;
                    inst->Internal.State = state_done;
                }
            }
            else{
                inst->ErrorID = error;
                inst->Error = 1;
                inst->Internal.State = state_error;
            }

            break;

        case state_done:

            if(!inst->Execute){
                inst->Done = 0;
                std::memset(reinterpret_cast<void*>(inst->Internal.DataAddress), 0, inst->Internal.DataSize);
                inst->Busy = 0;
                inst->Internal.State = state_idle;
            }

            break;

        case state_error:

            if(!inst->Execute){
                inst->ErrorID = ERR_OK;
                inst->Error = 0;
                inst->Busy = 0;
                inst->Internal.State = state_idle;
            }

            break;

    }

}
```

#### rl6dDestAddRecoveryPosFromData.cpp - rl6dRouterAddPathFromData Implementation
```cpp
#include "Router.hpp"

extern "C" _BUR_PUBLIC void rl6dDestAddRecoveryPosFromData(struct rl6dDestAddRecoveryPosFromData* inst){

    if(inst == nullptr){
        return;
    }

    Destination* d;
    std::shared_ptr<Destination> destination;
    rl6dPositionType* position;
    DINT error;

    enum state{
        state_idle,
        state_add_recovery_pos,
        state_done,
        state_error
    };

    switch(inst->Internal.State){

        case state_idle:

            if(inst->Execute){
                inst->Busy = 1;
                inst->Internal.State = state_add_recovery_pos;
            }

            break;

        case state_add_recovery_pos:

            error = check_destination_reference(inst->Destination);
            if(error == ERR_OK){
                if(inst->DataSize % sizeof(rl6dPositionType) != 0){
                    error = rl6dERR_DATA_ALIGNMENT;
                }
            }
            if(error == ERR_OK){
                d = reinterpret_cast<Destination*>(inst->Destination->Ident);
                destination = d->get_shared_ptr();
                if(destination->sem_acquire()){
                    for(UDINT offset = 0; offset < inst->DataSize; offset += sizeof(rl6dPositionType)){
                        position = reinterpret_cast<rl6dPositionType*>(inst->DataAddress + offset);
                        destination->add_recovery_position(*position);
                    }
                    destination->sem_release();
                    inst->Done = 1;
                    inst->Internal.State = state_done;
                }
            }
            else{
                inst->ErrorID = error;
                inst->Error = 1;
                inst->Internal.State = state_error;
            }
            break;

        case state_done:

            if(!inst->Execute){
                inst->Done = 0;
                inst->Busy = 0;
                inst->Internal.State = state_idle;
            }

            break;

        case state_error:

            if(!inst->Execute){
                inst->ErrorID = ERR_OK;
                inst->Error = 0;
                inst->Busy = 0;
                inst->Internal.State = state_idle;
            }

            break;
    }

}
```

#### rl6dDestinationSetWaypoint.cpp - rl6dWaypointSetNextWaypoint Implementation
```cpp
#include "Router.hpp"

extern "C" _BUR_PUBLIC void rl6dDestinationSetWaypoint(struct rl6dDestinationSetWaypoint* inst){

    if(inst == nullptr){
        return;
    }

    Destination* d;
    std::shared_ptr<Destination> destination;
    Waypoint* w;
    DINT error;

    enum state{
        state_idle,
        state_done,
        state_error
    };

    switch(inst->Internal.State){

        case state_idle:

            if(inst->Execute){
                inst->Busy = 1;
                error = check_destination_reference(inst->Destination);
                if(error == ERR_OK){
                    error = check_waypoint_reference(inst->Waypoint);
                }
                if(error == ERR_OK){
                    d = reinterpret_cast<Destination*>(inst->Destination->Ident);
                    destination = d->get_shared_ptr();
                    w = reinterpret_cast<Waypoint*>(inst->Waypoint->Ident);
                    destination->set_waypoint(w->get_shared_ptr());
                    inst->Done = 1;
                    inst->Internal.State = state_done;
                }
                else{
                    inst->ErrorID = error;
                    inst->Error = 1;
                    inst->Internal.State = state_error;
                }
            }

            break;

        case state_done:

            if(!inst->Execute){
                inst->Done = 0;
                inst->Busy = 0;
                inst->Internal.State = state_idle;
            }

            break;

        case state_error:

            if(!inst->Execute){
                inst->ErrorID = ERR_OK;
                inst->Error = 0;
                inst->Busy = 0;
                inst->Internal.State = state_idle;
            }

            break;
    }

}
```

#### rl6dWaypointAddDestination.cpp - rl6dWaypointAddDestination Implementation
```cpp
#include "Router.hpp"

extern "C" _BUR_PUBLIC void rl6dWaypointAddDestination(struct rl6dWaypointAddDestination* inst){

    if(inst == nullptr){
        return;
    }

    Waypoint* w;
    std::shared_ptr<Waypoint> waypoint;
    Destination* d;
    Path* p;
    std::shared_ptr<Path> path;
    DINT error;

    enum state{
        state_idle,
        state_add_destination,
        state_done,
        state_error
    };

    switch(inst->Internal.State){

        case state_idle:

            if(inst->Execute){
                inst->Busy = 1;
                inst->Internal.State = state_add_destination;
            }

            break;

        case state_add_destination:

            error = check_waypoint_reference(inst->Waypoint);
            if(error == ERR_OK){
                error = check_destination_reference(inst->Destination);
            }
            if((error == ERR_OK) && (inst->DeparturePath != nullptr)){
                error = check_path_reference(inst->DeparturePath);
            }
            if(error == ERR_OK){
                w = reinterpret_cast<Waypoint*>(inst->Waypoint->Ident);
                waypoint = w->get_shared_ptr();
                if(waypoint->sem_acquire()){
                    if(inst->DeparturePath != nullptr){
                        p = reinterpret_cast<Path*>(inst->Waypoint->Ident);
                        path = p->get_shared_ptr();
                    }
                    d = reinterpret_cast<Destination*>(inst->Destination->Ident);
                    waypoint->add_destination(d->get_shared_ptr(), path);
                    waypoint->sem_release();
                    inst->Done = 1;
                    inst->Internal.State = state_done;
                }
            }
            else{
                inst->ErrorID = error;
                inst->Error = 1;
                inst->Internal.State = state_error;
            }
            break;

        case state_done:

            if(!inst->Execute){
                inst->Done = 0;
                inst->Busy = 0;
                inst->Internal.State = state_idle;
            }

            break;

        case state_error:

            if(!inst->Execute){
                inst->ErrorID = ERR_OK;
                inst->Error = 0;
                inst->Busy = 0;
                inst->Internal.State = state_idle;
            }

            break;
    }

}
```

#### rl6dWaypointSetNextWaypoint.cpp - rl6dWaypointSetNextWaypoint Implementation
```cpp
#include "Router.hpp"

extern "C" _BUR_PUBLIC void rl6dWaypointSetNextWaypoint(struct rl6dWaypointSetNextWaypoint* inst){

    if(inst == nullptr){
        return;
    }

    Waypoint* w;
    std::shared_ptr<Waypoint> waypoint;
    Waypoint* w_n;
    DINT error;

    enum state{
        state_idle,
        state_done,
        state_error
    };

    switch(inst->Internal.State){

        case state_idle:

            if(inst->Execute){
                inst->Busy = 1;
                error = check_waypoint_reference(inst->Waypoint);
                if(error == ERR_OK){
                    error = check_waypoint_reference(inst->NextWaypoint);
                }
                if(error == ERR_OK){
                    w = reinterpret_cast<Waypoint*>(inst->Waypoint->Ident);
                    waypoint = w->get_shared_ptr();
                    w_n = reinterpret_cast<Waypoint*>(inst->NextWaypoint->Ident);
                    waypoint->set_next_waypoint(w_n->get_shared_ptr());
                    inst->Done = 1;
                    inst->Internal.State = state_done;
                }
                else{
                    inst->ErrorID = error;
                    inst->Error = 1;
                    inst->Internal.State = state_error;
                }
            }

            break;

        case state_done:

            if(!inst->Execute){
                inst->Done = 0;
                inst->Busy = 0;
                inst->Internal.State = state_idle;
            }

            break;

        case state_error:

            if(!inst->Execute){
                inst->ErrorID = ERR_OK;
                inst->Error = 0;
                inst->Busy = 0;
                inst->Internal.State = state_idle;
            }

            break;
    }

}
```

#### rl6dRouterAddShFromAsm.cpp - rl6dRouterAddShFromAsm Implementation
```cpp
#include "Router.hpp"

extern "C" _BUR_PUBLIC void rl6dRouterAddShFromAsm(struct rl6dRouterAddShFromAsm* inst){

    if(inst == nullptr){
        return;
    }

    Router* r;
    DINT error;

    enum state{
        state_idle,
        state_send_cmd,
        state_add_shuttles,
        state_done,
        state_error
    };

    switch(inst->Internal.State){

        case state_idle:

            if(inst->Execute){
                inst->Busy = 1;
                inst->Internal.State = state_send_cmd;
            }

            break;

        case state_send_cmd:

            error = check_router_reference(inst->Router);
            if(error == ERR_OK){
                r = reinterpret_cast<Router*>(inst->Router->Ident);
                if(r->get_initialized()){
                    if(r->acquire_cmd_semaphore()){
                        if(r->get_cmd_ready()){
                            r->set_add_sh_from_asm();
                            inst->Internal.State = state_add_shuttles;
                        }
                        else{
                            r->release_cmd_semaphore();
                        }
                    }
                }
            }
            else{
                inst->ErrorID  = error;
                inst->Error = 1;
                inst->Internal.State = state_error;
            }

            break;

        case state_add_shuttles:

            error = check_router_reference(inst->Router);
            if(error == ERR_OK){
                r = reinterpret_cast<Router*>(inst->Router->Ident);
                if(r->get_done()){
                    inst->NumShuttles = r->get_num_asm_sh();
                    r->reset_add_sh_from_asm();
                    r->release_cmd_semaphore();
                    inst->Done = 1;
                    inst->Internal.State = state_done;
                }
                else if(r->get_error()){
                    r->reset_add_sh_from_asm();
                    inst->ErrorID  = r->get_error_id();
                    inst->Error = 1;
                    r->set_error_reset();
                    r->release_cmd_semaphore();
                    inst->Internal.State = state_error;
                }
            }
            else{
                inst->ErrorID  = error;
                inst->Error = 1;
                inst->Internal.State = state_error;
            }

            break;

        case state_done:

            if(!inst->Execute){
                inst->Done = 0;
                inst->Busy = 0;
                inst->NumShuttles = 0;
                inst->Internal.State = state_idle;
            }

            break;

        case state_error:

            if(!inst->Execute){
                inst->ErrorID = ERR_OK;
                inst->Error = 0;
                inst->Busy = 0;
                inst->Internal.State = state_idle;
            }

            break;

    }

}
```

#### rl6dRouterExecuteRecovery.cpp - rl6dRouterExecuteRecovery Implementation
```cpp
#include "Router.hpp"

extern "C" _BUR_PUBLIC void rl6dRouterExecuteRecovery(struct rl6dRouterExecuteRecovery* inst){

    if(inst == nullptr){
        return;
    }

    Router* r;
    DINT error;

    enum state{
        state_idle,
        state_send_cmd,
        state_recover,
        state_done,
        state_error
    };

    switch(inst->Internal.State){

        case state_idle:

            if(inst->Execute){
                inst->Busy = 1;
                inst->Internal.State = state_send_cmd;
            }

            break;

        case state_send_cmd:

            error = check_router_reference(inst->Router);
            if(error == ERR_OK){
                r = reinterpret_cast<Router*>(inst->Router->Ident);
                if(r->get_initialized()){
                    if(r->acquire_cmd_semaphore()){
                        if(r->get_cmd_ready()){
                            r->set_recover_shuttles(inst->Mode, inst->Velocity, inst->Acceleration);
                            inst->Internal.State = state_recover;
                        }
                        else{
                            r->release_cmd_semaphore();
                        }
                    }
                }
            }
            else{
                inst->ErrorID  = error;
                inst->Error = 1;
                inst->Internal.State = state_error;
            }

            break;

        case state_recover:

            error = check_router_reference(inst->Router);
            if(error == ERR_OK){
                r = reinterpret_cast<Router*>(inst->Router->Ident);
                if(r->get_done()){
                    r->reset_recover_shuttles();
                    r->release_cmd_semaphore();
                    inst->Done = 1;
                    inst->Internal.State = state_done;
                }
                else if(r->get_error()){
                    r->reset_recover_shuttles();
                    inst->ErrorID  = r->get_error_id();
                    inst->Error = 1;
                    r->set_error_reset();
                    r->release_cmd_semaphore();
                    inst->Internal.State = state_error;
                }
            }
            else{
                inst->ErrorID  = error;
                inst->Error = 1;
                inst->Internal.State = state_error;
            }

            break;

        case state_done:

            if(!inst->Execute){
                inst->Done = 0;
                inst->Busy = 0;
                inst->Internal.State = state_idle;
            }

            break;

        case state_error:

            if(!inst->Execute){
                inst->ErrorID = ERR_OK;
                inst->Error = 0;
                inst->Busy = 0;
                inst->Internal.State = state_idle;
            }

            break;

    }

}
```

#### rl6dDestinationMonitor.cpp - rl6dDestinationMonitor Implementation
```cpp
#include "Router.hpp"

extern "C" _BUR_PUBLIC void rl6dDestinationMonitor(struct rl6dDestinationMonitor* inst){

    if(inst == nullptr){
        return;
    }

    Destination* d;
    std::shared_ptr<Destination> destination;
    DestinationIf* i;
    std::shared_ptr<DestinationIf> interface;
    std::shared_ptr<Shuttle> shuttle;
    DINT error;

    enum state{
        state_idle,
        state_get_interface,
        state_wait_shuttle,
        state_wait_not_acknowledge,
        state_wait_acknowledge,
        state_error
    };

    switch(inst->Internal.State){

        case state_idle:

            if(inst->Enable){
                inst->Busy = 1;
                inst->Internal.State = state_get_interface;
            }

            break;

        case state_get_interface:

            error = check_destination_reference(inst->Destination);
            if(error == ERR_OK){
                d = reinterpret_cast<Destination*>(inst->Destination->Ident);
                destination = d->get_shared_ptr();
                if(destination->sem_acquire()){
                    inst->Internal.Reference = reinterpret_cast<std::uintptr_t>(destination->create_interface().get());
                    destination->sem_release();
                    inst->Internal.State = state_wait_shuttle;
                }
            }
            else{
                inst->ErrorID = error;
                inst->Error = 1;
                inst->Internal.State = state_error;
            }

            break;

        case state_wait_shuttle:

            error = check_destination_if_reference(inst->Internal.Reference);
            if(error == ERR_OK){
                if(inst->Enable){
                    i = reinterpret_cast<DestinationIf*>(inst->Internal.Reference);
                    interface = i->get_shared_ptr();
                    if(interface->shuttle_is_present()){
                        shuttle = interface->get_shuttle_present().lock();
                        inst->ShuttleID = shuttle->get_shuttle_id();
                        inst->RouterShuttle.Ident = reinterpret_cast<std::uintptr_t>(shuttle.get());
                        inst->Mc6DShuttle = *shuttle->get_shuttle_reference();
                        inst->ShuttlePresent = 1;
                        interface->acknowledge_shuttle();
                        if(inst->AcknowledgeShuttle){
                            inst->Internal.State = state_wait_not_acknowledge;
                        }
                        else{
                            inst->Internal.State = state_wait_acknowledge;
                        }
                    }
                    inst->Valid = 1;
                }
                else{
                    i = reinterpret_cast<DestinationIf*>(inst->Internal.Reference);
                    interface = i->get_shared_ptr();
                    interface->set_delete();
                    inst->Valid = 0;
                    inst->ShuttlePresent = 0;
                    inst->ShuttleID = 0;
                    std::memset(&inst->Mc6DShuttle, 0, sizeof(inst->Mc6DShuttle));
                    std::memset(&inst->RouterShuttle, 0, sizeof(inst->RouterShuttle));
                    inst->Busy = 0;
                    inst->Internal.State = state_idle;
                }
            }
            else{
                inst->ErrorID = error;
                inst->Error = 1;
                inst->Internal.State = state_error;
            }

            break;

        case state_wait_not_acknowledge:

            if(inst->Enable){
                if(!inst->AcknowledgeShuttle){
                    inst->Internal.State = state_wait_acknowledge;
                }
            }
            else{
                error = check_destination_if_reference(inst->Internal.Reference);
                if(error == ERR_OK){
                    i = reinterpret_cast<DestinationIf*>(inst->Internal.Reference);
                    interface = i->get_shared_ptr();
                    interface->set_delete();
                    inst->Valid = 0;
                    inst->ShuttlePresent = 0;
                    inst->ShuttleID = 0;
                    std::memset(&inst->Mc6DShuttle, 0, sizeof(inst->Mc6DShuttle));
                    std::memset(&inst->RouterShuttle, 0, sizeof(inst->RouterShuttle));
                    inst->Busy = 0;
                    inst->Internal.State = state_idle;
                }
                else{
                    inst->Valid = 0;
                    inst->ShuttlePresent = 0;
                    inst->ShuttleID = 0;
                    std::memset(&inst->Mc6DShuttle, 0, sizeof(inst->Mc6DShuttle));
                    std::memset(&inst->RouterShuttle, 0, sizeof(inst->RouterShuttle));
                    inst->ErrorID = error;
                    inst->Error = 1;
                    inst->Internal.State = state_error;
                }
            }

            break;

        case state_wait_acknowledge:

            if(inst->Enable){
                if(inst->AcknowledgeShuttle){
                    inst->ShuttlePresent = 0;
                    inst->ShuttleID = 0;
                    std::memset(&inst->Mc6DShuttle, 0, sizeof(inst->Mc6DShuttle));
                    std::memset(&inst->RouterShuttle, 0, sizeof(inst->RouterShuttle));
                    inst->Internal.State = state_wait_shuttle;
                }
            }
            else{
                error = check_destination_if_reference(inst->Internal.Reference);
                if(error == ERR_OK){
                    i = reinterpret_cast<DestinationIf*>(inst->Internal.Reference);
                    interface = i->get_shared_ptr();
                    interface->set_delete();
                    inst->Valid = 0;
                    inst->ShuttlePresent = 0;
                    inst->ShuttleID = 0;
                    std::memset(&inst->Mc6DShuttle, 0, sizeof(inst->Mc6DShuttle));
                    std::memset(&inst->RouterShuttle, 0, sizeof(inst->RouterShuttle));
                    inst->Busy = 0;
                    inst->Internal.State = state_idle;
                }
                else{
                    inst->Valid = 0;
                    inst->ShuttlePresent = 0;
                    inst->ShuttleID = 0;
                    std::memset(&inst->Mc6DShuttle, 0, sizeof(inst->Mc6DShuttle));
                    std::memset(&inst->RouterShuttle, 0, sizeof(inst->RouterShuttle));
                    inst->ErrorID = error;
                    inst->Error = 1;
                    inst->Internal.State = state_error;
                }
            }

            break;

        case state_error:

            if(!inst->Enable){
                inst->ErrorID = ERR_OK;
                inst->Error = 0;
                inst->Busy = 0;
                inst->Internal.State = state_idle;
            }

            break;

    }

}
```

#### rl6dShuttleMoveDestination.cpp - rl6dDestinationMonitor Implementation
```cpp
#include "Router.hpp"

extern "C" _BUR_PUBLIC void rl6dShuttleMoveDestination(struct rl6dShuttleMoveDestination* inst){

    if(inst == nullptr){
        return;
    }

    Destination* d;
    std::shared_ptr<Destination> destination;
    Waypoint* w;
    std::weak_ptr<Waypoint> waypoint;
    Shuttle* s;
    std::shared_ptr<Shuttle> shuttle;
    ShuttleIf* i;
    std::shared_ptr<ShuttleIf> interface;
    DINT error;

    enum state{
        state_idle,
        state_send_cmd,
        state_move,
        state_done,
        state_error
    };

    switch(inst->Internal.State){

        case state_idle:

            if(inst->Execute){
                inst->Busy = 1;
                inst->Internal.State = state_send_cmd;
            }

            break;

        case state_send_cmd:

            error = check_shuttle_reference(inst->RouterShuttle);
            if(error == ERR_OK){
                error = check_destination_reference(inst->Destination);
            }
            if(error == ERR_OK){
                s = reinterpret_cast<Shuttle*>(inst->RouterShuttle->Ident);
                shuttle = s->get_shared_ptr();
                if(shuttle->sem_acquire()){
                    inst->Internal.Reference = reinterpret_cast<std::uintptr_t>(shuttle->create_interface().get());
                    shuttle->sem_release();
                    d = reinterpret_cast<Destination*>(inst->Destination->Ident);
                    destination = d->get_shared_ptr();
                    error = check_shuttle_if_reference(inst->Internal.Reference);
                    if(error == ERR_OK){
                        i = reinterpret_cast<ShuttleIf*>(inst->Internal.Reference);
                        interface = i->get_shared_ptr();
                        if (inst->Waypoint != nullptr){
                            error = check_waypoint_reference(inst->Waypoint);
                            if(error == ERR_OK){
                                w = reinterpret_cast<Waypoint*>(inst->Waypoint->Ident);
                                waypoint = w->get_shared_ptr();
                                interface->set_destination_waypoint(destination, waypoint, inst->Velocity, inst->Acceleration);
                                inst->Internal.State = state_move;
                            }
                            else{
                                inst->ErrorID = error;
                                inst->Error = 1;
                                inst->Internal.State = state_error;
                            }
                        }
                        else{
                            interface->set_destination(destination, inst->Velocity, inst->Acceleration);
                            inst->Internal.State = state_move;
                        }
                    }
                    else{
                        inst->ErrorID = error;
                        inst->Error = 1;
                        inst->Internal.State = state_error;
                    }
                }
            }
            else{
                inst->ErrorID = error;
                inst->Error = 1;
                inst->Internal.State = state_error;
            }

            break;

        case state_move:

            error = check_shuttle_if_reference(inst->Internal.Reference);
            if(error == ERR_OK){
                i = reinterpret_cast<ShuttleIf*>(inst->Internal.Reference);
                interface = i->get_shared_ptr();
                if(inst->Execute){
                    if(interface->get_error()){
                        inst->ErrorID = interface->get_error_id();
                        inst->Error = 1;
                        inst->Active = 0;
                        inst->Aborted = 0;
                        inst->Done = 0;
                        inst->Internal.State = state_error;
                    }
                    else{
                        inst->Active = interface->get_move_active();
                        inst->Aborted = interface->get_aborted();
                        inst->Done = interface->get_move_done();
                    }
                }
                else{
                    inst->Active = 0;
                    inst->Aborted = 0;
                    inst->Done = 0;
                    interface->set_delete();
                    inst->Internal.Reference = 0;
                    inst->Busy = 0;
                    inst->Internal.State = state_idle;
                }
            }
            else{
                inst->Active = 0;
                inst->Aborted = 0;
                inst->Done = 0;
                inst->ErrorID = error;
                inst->Error = 1;
                inst->Internal.State = state_error;
            }

            break;

        case state_error:

            if(!inst->Execute){
                error = check_shuttle_if_reference(inst->Internal.Reference);
                if(error == ERR_OK){
                    interface->set_delete();
                    inst->Internal.Reference = 0;
                }
                inst->ErrorID = ERR_OK;
                inst->Error = 0;
                inst->Busy = 0;
                inst->Internal.State = state_idle;
            }

            break;

    }

}
```

#### rl6dShCopyUserData.cpp - rl6dShCopyUserData Implementation
```cpp
#include "Shuttle.hpp"
#include "CheckRef.hpp"

extern "C" _BUR_PUBLIC void rl6dShCopyUserData(struct rl6dShCopyUserData* inst){

    if(inst == nullptr){
        return;
    }

    Shuttle* s;
    std::shared_ptr<Shuttle> shuttle;
    DINT error;

    enum state{
        state_idle,
        state_done,
        state_error
    };

    switch(inst->Internal.State){

        case state_idle:

            if(inst->Execute){
                inst->Busy = 1;
                error = check_shuttle_reference(inst->RouterShuttle);
                if(error == ERR_OK){
                    if(inst->DataAddress == 0){
                        error = rl6dERR_USER_DATA_NULL_POINTER;
                    }
                }
                if(error == ERR_OK){
                    if(inst->DataSize == 0){
                        error = rl6dERR_USER_DATA_SIZE_ZERO;
                    }
                }
                if(error == ERR_OK){
                    s = reinterpret_cast<Shuttle*>(inst->RouterShuttle->Ident);
                    shuttle = s->get_shared_ptr();
                    ReadUserDataResult result = shuttle->read_user_data();
                    if(result.size == inst->DataSize){
                        if(inst->Mode == rl6dSH_COPY_USER_DATA_READ){
                            std::memcpy(reinterpret_cast<char*>(inst->DataAddress), result.value, result.size);
                            inst->SizeCopied = result.size;
                        }
                        else if(inst->Mode == rl6dSH_COPY_USER_DATA_WRITE){
                            inst->SizeCopied = shuttle->write_user_data(reinterpret_cast<char*>(inst->DataAddress), inst->DataSize);
                        }
                        inst->Done = 1;
                        inst->Internal.State = state_done;
                    }
                    else{
                        inst->ErrorID = rl6dERR_USER_DATA_SIZE_MISMATCH;
                        inst->Error = 1;
                        inst->Internal.State = state_error;
                    }
                }
                else{
                    inst->ErrorID = error;
                    inst->Error = 1;
                    inst->Internal.State = state_error;
                }
            }

            break;

        case state_done:

            if(!inst->Execute){
                inst->Done = 0;
                inst->SizeCopied = 0;
                inst->Busy = 0;
                inst->Internal.State = state_idle;
            }

            break;

        case state_error:

            if(!inst->Execute){
                inst->ErrorID = ERR_OK;
                inst->Error = 0;
                inst->Busy = 0;
                inst->Internal.State = state_idle;
            }

            break;

    }

}
```

#### rl6dShCopyUserDataSync.cpp - rl6dShCopyUserDataSync Implementation
```cpp
#include "Shuttle.hpp"
#include "CheckRef.hpp"

extern "C" _BUR_PUBLIC signed long rl6dShCopyUserDataSync(struct rl6dShuttleType* RouterShuttle, enum rl6dShCopyUserDataModeEnum Mode, unsigned long DataAddress, unsigned long DataSize){

    Shuttle* s;
    std::shared_ptr<Shuttle> shuttle;
    DINT error;

    error = check_shuttle_reference(RouterShuttle);
    if(error == ERR_OK){
        if(DataAddress == 0){
            error = rl6dERR_USER_DATA_NULL_POINTER;
        }
    }
    if(error == ERR_OK){
        if(DataSize == 0){
            error = rl6dERR_USER_DATA_SIZE_ZERO;
        }
    }
    if(error == ERR_OK){
        s = reinterpret_cast<Shuttle*>(RouterShuttle->Ident);
        shuttle = s->get_shared_ptr();
        ReadUserDataResult result = shuttle->read_user_data();
        if(result.size == DataSize){
            if(Mode == rl6dSH_COPY_USER_DATA_READ){
                std::memcpy(reinterpret_cast<char*>(DataAddress), result.value, DataSize);
            }
            else if(Mode == rl6dSH_COPY_USER_DATA_WRITE){
                shuttle->write_user_data(reinterpret_cast<char*>(DataAddress), DataSize);
            }
        }
        else{
            error = rl6dERR_USER_DATA_SIZE_MISMATCH;
        }
    }

    return error;

}
```

### Program Logical/Source/Core/RDICore (IEC)
